// TIA Portal V20 export
// export: Created 2026-08-17T22:42:35.3963519Z, ExportSetting None, DisplayName Totally Integrated Automation Portal, DisplayVersion V20 Update 3, DisplayName TIA Portal Openness, DisplayVersion V20 Update 3, DisplayName TIA Portal Version Control Interface, DisplayVersion V20 Update 3, DisplayName STEP 7 Professional, DisplayVersion V20 Update 3, DisplayName STEP 7 Safety, DisplayVersion V20 Update 2, DisplayName WinCC Basic/Comfort/Advanced, DisplayVersion V20 Update 3, DisplayName SIMATIC Visualization Architect, DisplayVersion V20 Update 3, DisplayName WinCC Unified, DisplayVersion V20 Update 3, DisplayName SIMATIC Visualization Architect, DisplayVersion V20 Update 3
FUNCTION_BLOCK "EM_TransferDischarge"   // FB15, LAD
{ S7_Optimized_Access := 'TRUE' }
// stored: MemoryReserve 100, SetENOAutomatically false
BEGIN
END_FUNCTION_BLOCK
